FUNCTION TrackingDifferentiator :LREAL

VAR_INPUT
	expect:LREAL;
END_VAR

v1 := v1 + ADRC_TD_h0 * v2;//跟新最速跟踪状态量x1
v2 := v2 + ADRC_TD_h0 * (-ADRC_TD_r0 * Sign(v1 - expect + (v2 * ABS(v2))/(2 * ADRC_TD_r0)));//跟新最速跟踪状态量微分x2

END_FUNCTION

(* stored: Version 1.1.0.1, ProductVersion 3.1.4024.11
   POU TrackingDifferentiator: Id {ec373d2a-a4bc-40dc-87dc-df17586bf4df}, SpecialFunc None *)
